TYPE ST_PowerMeasurement_status :
STRUCT
	b_RotaryField	: BOOL;
	b_GeneralWarning: BOOL;
	b_GeneralFault	: BOOL;
	b_OverVoltage 	: BOOL;
	b_UnderVoltage	: BOOL;
	b_OverCurrent	: BOOL;
	b_Error_Phase 	: ARRAY [1..3] OF BOOL;
END_STRUCT
END_TYPE

(* stored: Version 1.1.0.1, ProductVersion 3.1.4024.12
   DUT ST_PowerMeasurement_status: Id {ae5e65f1-a1c2-4cb1-b8c6-88483d39f239} *)
